# EPICS substitutions: src/test/ioc/X/MTEST-PC-JCAE/MTEST-PC-JCAE_test.subs
file test.template {
    {
        P = MTEST-PC-JCAE:
    }
}
